// TIA Portal V18 export
FUNCTION "TEMPLATE--v1.0--07_Speed Control" : Void   // FC24, F_LAD
TITLE = Manage Safety Encoder
{ S7_Optimized_Access := 'TRUE' }
// v1.0 First Emission
BEGIN

REGION Network 1: !!NetworkComment$$
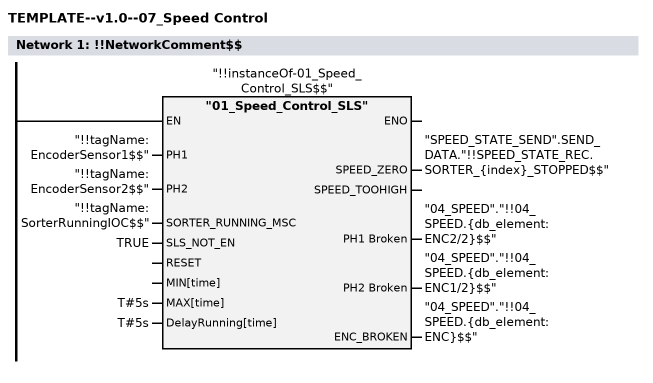
   RUNG wire#powerrail
      "!!instanceOf-01_Speed_Control_SLS$$"(PH1 := "!!tagName:EncoderSensor1$$", PH2 := "!!tagName:EncoderSensor2$$", SORTER_RUNNING_MSC := "!!tagName:SorterRunningIOC$$", SLS_NOT_EN := TRUE, RESET :=, "MIN[time]" :=, "MAX[time]" := T#5s, "DelayRunning[time]" := T#5s, SPEED_ZERO => "SPEED_STATE_SEND".SEND_DATA."!!SPEED_STATE_REC.SORTER_{index}_STOPPED$$", SPEED_TOOHIGH =>, "PH1 Broken" => "04_SPEED"."!!04_SPEED.{db_element:ENC2/2}$$", "PH2 Broken" => "04_SPEED"."!!04_SPEED.{db_element:ENC1/2}$$", ENC_BROKEN => "04_SPEED"."!!04_SPEED.{db_element:ENC}$$")
   END_RUNG
   // the same network as SCL:
   "!!instanceOf-01_Speed_Control_SLS$$"(PH1 := "!!tagName:EncoderSensor1$$",   // "01_Speed_Control_SLS"
                           PH2 := "!!tagName:EncoderSensor2$$",
                           SORTER_RUNNING_MSC := "!!tagName:SorterRunningIOC$$",
                           SLS_NOT_EN := TRUE,
                           "MAX[time]" := T#5s,
                           "DelayRunning[time]" := T#5s,
                           SPEED_ZERO => "SPEED_STATE_SEND".SEND_DATA."!!SPEED_STATE_REC.SORTER_{index}_STOPPED$$",
                           "PH1 Broken" => "04_SPEED"."!!04_SPEED.{db_element:ENC2/2}$$",
                           "PH2 Broken" => "04_SPEED"."!!04_SPEED.{db_element:ENC1/2}$$",
                           ENC_BROKEN => "04_SPEED"."!!04_SPEED.{db_element:ENC}$$");
END_REGION
END_FUNCTION
